PROGRAM WheelEncoders
VAR
zaehler : UINT := 0;


encDataOldMotor1:UINT:=0;
encDataOldMotor2:UINT:=0;
encDataOldMotor3:UINT:=0;

//Koordinatentransformation Weg
skalEnc:LREAL:=0.00766990393;

//Koordinatentransformation Geschwindigkeit
v1:LREAL:=0;
v2:LREAL:=0;
v3:LREAL:=0;
velocityFromMotor1:LREAL:=0;
velocityFromMotor2:LREAL:=0;
velocityFromMotor3:LREAL:=0;

//INPUTS
encDataFromMotor1 AT%I*  :UINT:=0;
encDataFromMotor2 AT%I*  :UINT:=0;
encDataFromMotor3 AT%I*  :UINT:=0;

diff1: INT := 0;
diff2: INT := 0;
diff3: INT := 0;

//OUTPUTS
veloFromMotors : RobotPose;

vXCartesianFromMotors AT%Q*:LREAL:=0;
vYCartesianFromMotors AT%Q*:LREAL:=0;
vthetaCartesianFromMotors AT%Q*:LREAL:=0;
END_VAR

IF DrehzahlRegler.state = CoreDriveState.Init THEN
	encDataOldMotor1 := encDataFromMotor1;
	encDataOldMotor2 := encDataFromMotor2;
	encDataOldMotor3 := encDataFromMotor3;
	//get ciyclictime of task

END_IF

// Encoder Wegberechnung und Differenzierung für Geschwindigkeit
diff1:=UINT_TO_INT(encDataFromMotor1) - UINT_TO_INT(encDataOldMotor1);
IF diff1 >= 32767 OR diff1 <= -32767 THEN
	diff1 := 0;
	zaehler := zaehler + 1;
END_IF
diff2:=UINT_TO_INT(encDataFromMotor2) - UINT_TO_INT(encDataOldMotor2);
IF diff2 >= 32767 OR diff2 <= -32767 THEN
	diff2 := 0;
END_IF
diff3:=UINT_TO_INT(encDataFromMotor3) - UINT_TO_INT(encDataOldMotor3);
IF diff3 >= 32767 OR diff3 <= -32767 THEN
	diff3 := 0;
END_IF

velocityFromMotor1:=diff1/DrehzahlRegler.diffConst*skalEnc;
velocityFromMotor2:=diff2/DrehzahlRegler.diffConst*skalEnc;
velocityFromMotor3:=diff3/DrehzahlRegler.diffConst*skalEnc;

// Koordinatentransformation Geschwindigkeit
v1:=-velocityFromMotor1;
v2:=-velocityFromMotor2;
v3:=-velocityFromMotor3;

vXCartesianFromMotors:=(v3 - v1) / (2.0 * COS(30.0*PI/180));  //in mm / s
vYCartesianFromMotors:=(v1 - 2.0 * v2 + v3) / 3.0;            //in mm / s
vThetaCartesianFromMotors:=(v1 + v2 + v3) / (3.0 * 135.0);    //in rad / s

veloFromMotors.x := vXCartesianFromMotors;
veloFromMotors.y := vYCartesianFromMotors;
veloFromMotors.theta := vThetaCartesianFromMotors;

// Alte Encoderdaten speichern
encDataOldMotor1:=encDataFromMotor1;
encDataOldMotor2:=encDataFromMotor2;
encDataOldMotor3:=encDataFromMotor3;

Main.setIstVeloEnc(VeloFromMotors);

END_PROGRAM

(* stored: Version 1.1.0.1, ProductVersion 3.1.4024.11
   POU WheelEncoders: Id {e5336efa-79c2-40d6-9ef7-789a94ea11a6}, SpecialFunc None *)
